FUNCTION_BLOCK fbInverterJogCtrl
VAR_INPUT
	bEnable			: BOOL;
	bEmergencyStop	: BOOL;
	bLeftOT			: BOOL;
	bRightOT		: BOOL;
	bArmJogFor		: BOOL;
	bArmJogRev		: BOOL;
	iJogRPM		: INT;
	rRatio			: REAL;

END_VAR
VAR_OUTPUT
	bMoveForFlag	: BOOL;
	bMoveRevFlag	: BOOL;
END_VAR

VAR_IN_OUT
	iMoveRPM		: INT;

END_VAR
VAR
	LeftOtAlarm: BOOL;
	RightOtAlarm: BOOL;
	JogForFb: AM_InverterConversionHz;
	iMoveRPMTemp: INT;
END_VAR
VAR // added by the converter: edge detectors and wires of the graphical bodies
    _w1, _w2 : INT;
END_VAR

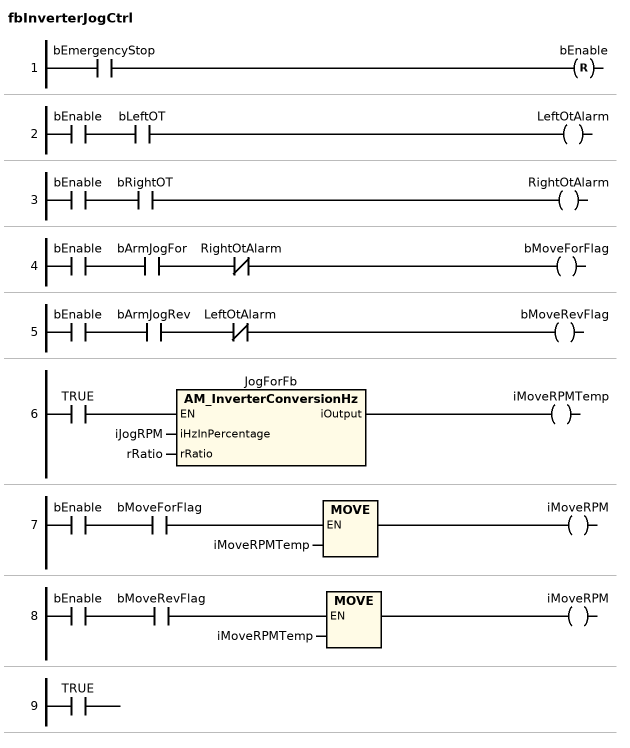
// NETWORK 1
bEnable R= bEmergencyStop;

// NETWORK 2
LeftOtAlarm := bEnable AND bLeftOT;

// NETWORK 3
RightOtAlarm := bEnable AND bRightOT;

// NETWORK 4
bMoveForFlag := bEnable AND bArmJogFor AND NOT RightOtAlarm;

// NETWORK 5
bMoveRevFlag := bEnable AND bArmJogRev AND NOT LeftOtAlarm;

// NETWORK 6
JogForFb(iHzInPercentage := iJogRPM, rRatio := rRatio); // AM_InverterConversionHz
iMoveRPMTemp := JogForFb.iOutput;

// NETWORK 7
IF bEnable AND bMoveForFlag THEN _w1 := iMoveRPMTemp; END_IF
iMoveRPM := _w1;

// NETWORK 8
IF bEnable AND bMoveRevFlag THEN _w2 := iMoveRPMTemp; END_IF
iMoveRPM := _w2;

// NETWORK 9

END_FUNCTION_BLOCK

(* stored: Version 1.1.0.1, ProductVersion 3.1.4024.12
   POU fbInverterJogCtrl: Id {36c96843-c88a-4860-aaf2-a3a63cadd327}, SpecialFunc None *)
